FUNCTION_BLOCK AxisHaltTestSuite
VAR
	StubAxis : AXIS_REF;
	TestAxisHalt : Mc2Halt(StubAxis);
	ReRun: BOOL;
END_VAR

DoesTaskRejectHaltWhenStationary();
IF ReRun THEN
	TestSuite.ReRunTests();
	ReRun := FALSE;
END_IF

METHOD DoesTaskRejectHaltWhenStationary : BOOL
VAR_INST
	Expected : HRESULT;
	Actual	 : HRESULT;
END_VAR
IF TestSuite.Test(__POUNAME()).ExecuteTest() THEN
	Expected := S_FALSE;
	Actual := TestAxisHalt.Execute();
	TestSuite.Test(__POUNAME()).AssertEqual(Expected, Actual);
END_IF
END_METHOD

END_FUNCTION_BLOCK

(* stored: Version 1.1.0.1
   POU AxisHaltTestSuite: Id {506c244a-6b71-4d33-aeec-65d4d3cf5d5e}, SpecialFunc None
   Method DoesTaskRejectHaltWhenStationary: Id {d10470f1-6c20-4eed-b536-d69117943531} *)
